FUNCTION_BLOCK FB_Button

VAR
	byButtonInput AT %I* : BIT;
	byButtonLight AT %Q* : BIT;
END_VAR

METHOD mButtonLight : BOOL

VAR_INPUT
	//byButtonInput : BYTE;
END_VAR

IF byButtonInput THEN
	byButtonLight := TRUE;

ELSE
	byButtonLight := FALSE;
END_IF
END_METHOD

END_FUNCTION_BLOCK

(* stored: Version 1.1.0.1, ProductVersion 3.1.4024.12
   POU FB_Button: Id {fd94e3b4-70ec-498d-97ca-45a1e18c22a5}, SpecialFunc None
   Method mButtonLight: Id {e941f189-7ebc-474d-9333-65e91250941f} *)
